// TIA Portal V16 export
// export: Created 2019-09-22T11:06:18.3137336Z, ExportSetting WithDefaults, DisplayName Totally Integrated Automation Portal, DisplayVersion V16, DisplayName TIA Portal Version Control Interface, DisplayVersion V16, DisplayName TIA Portal Openness, DisplayVersion V16, DisplayName STEP 7 Professional, DisplayVersion V16, DisplayName SIMATIC Energy Suite, DisplayVersion V16, DisplayName STEP 7 Safety, DisplayVersion V16, DisplayName WinCC Professional, DisplayVersion V16, DisplayName SIMATIC Visualization Architect, DisplayVersion V16
DATA_BLOCK "InstDiagStartupIoSystem1"   // DB2001
VERSION : 0.1
// stored: AutoNumber true, InstanceOfName DiagStartupIoSystem, InstanceOfType FB
"DiagStartupIoSystem"
   // VAR_INPUT
   //    ioSystemHwId : HW_IOSYSTEM;
   // END_VAR
   // VAR_OUTPUT
   //    status : Int;
   //    instructionError : Int;
   //    errorIndex : Int;
   // END_VAR
   // VAR_IN_OUT
   //    ioSystem : "typeIoSystem";
   // END_VAR
   // VAR
   //    statActualConfiguredDevices : Int;
   //    statGeoAddr { ExternalAccessible := 'False'; ExternalVisible := 'False'; ExternalWritable := 'False'; S7_SetPoint := 'True'} : GEOADDR;
   //    statGeoLaddr { ExternalAccessible := 'False'; ExternalVisible := 'False'; ExternalWritable := 'False'} : HW_ANY;
   //    statConfiguredDevices { ExternalAccessible := 'False'; ExternalVisible := 'False'; ExternalWritable := 'False'} : Array[0..1023] of Bool;
   //    statExistingDevices : Array[0..1023] of Bool;
   //    statFaultyDevices : Array[0..1023] of Bool;
   //    statDisabledDevices { ExternalAccessible := 'False'; ExternalVisible := 'False'; ExternalWritable := 'False'} : Array[0..1023] of Bool;
   //    statProblemDevices { ExternalAccessible := 'False'; ExternalVisible := 'False'; ExternalWritable := 'False'} : Array[0..1023] of Bool;
   //    statDeviceModuleStates : Array[0..127] of Bool;
   //    instGetNameDevices { S7_SetPoint := 'True'} : Get_Name;
   //    statInitString : String;
   //    statFirstDevice : UInt;
   //    statFirstDeviceFlag { ExternalAccessible := 'False'; ExternalVisible := 'False'; ExternalWritable := 'False'} : Bool;
   //    statLastDevice : UInt;
   //    statLinkedListPointer : Int;
   //    statFirstRun : Bool;
   //    statResetStatesOld : Bool;
   //    statMaxDevices : Int;
   // END_VAR
BEGIN
END_DATA_BLOCK
